(* PLC project LTAB4, Bombardier Transportation 1131-TOOL 3.1.0.1 *)
(* stored: companyURL www.kw-software.com, creationDateTime 2014-05-22T08:06:31, version 1400738791, modificationDateTime 2014-05-22T08:06:31 *)

FUNCTION_BLOCK DBC_PV_MtFanCtrl
  VAR_INPUT
    DBC_PV_X_ColStep : INT;
  END_VAR
  VAR_OUTPUT
    DBC_PV_C_Fan1Lo : BOOL;
    DBC_PV_C_Fan1Hi : BOOL;
    DBC_PV_C_Fan2Lo : BOOL;
    DBC_PV_C_Fan2Hi : BOOL;
    DBC_PV_C_Fan3Lo : BOOL;
    DBC_PV_C_Fan3Hi : BOOL;
  END_VAR
  VAR
    Enable : BOOL := TRUE;
    P_Fan1Lo_1 : INT := 3;
    P_Fan1Lo_2 : INT := 7;
    P_Fan1Hi : INT := 8;
    P_Fan2Lo_1 : INT := 4;
    P_Fan2Lo_2 : INT := 6;
    P_Fan2Hi_1 : INT := 7;
    P_Fan2Hi_2 : INT := 8;
    P_Fan3Lo : INT := 5;
    P_Fan3Hi_1 : INT := 6;
    P_Fan3Hi_2 : INT := 8;
  END_VAR

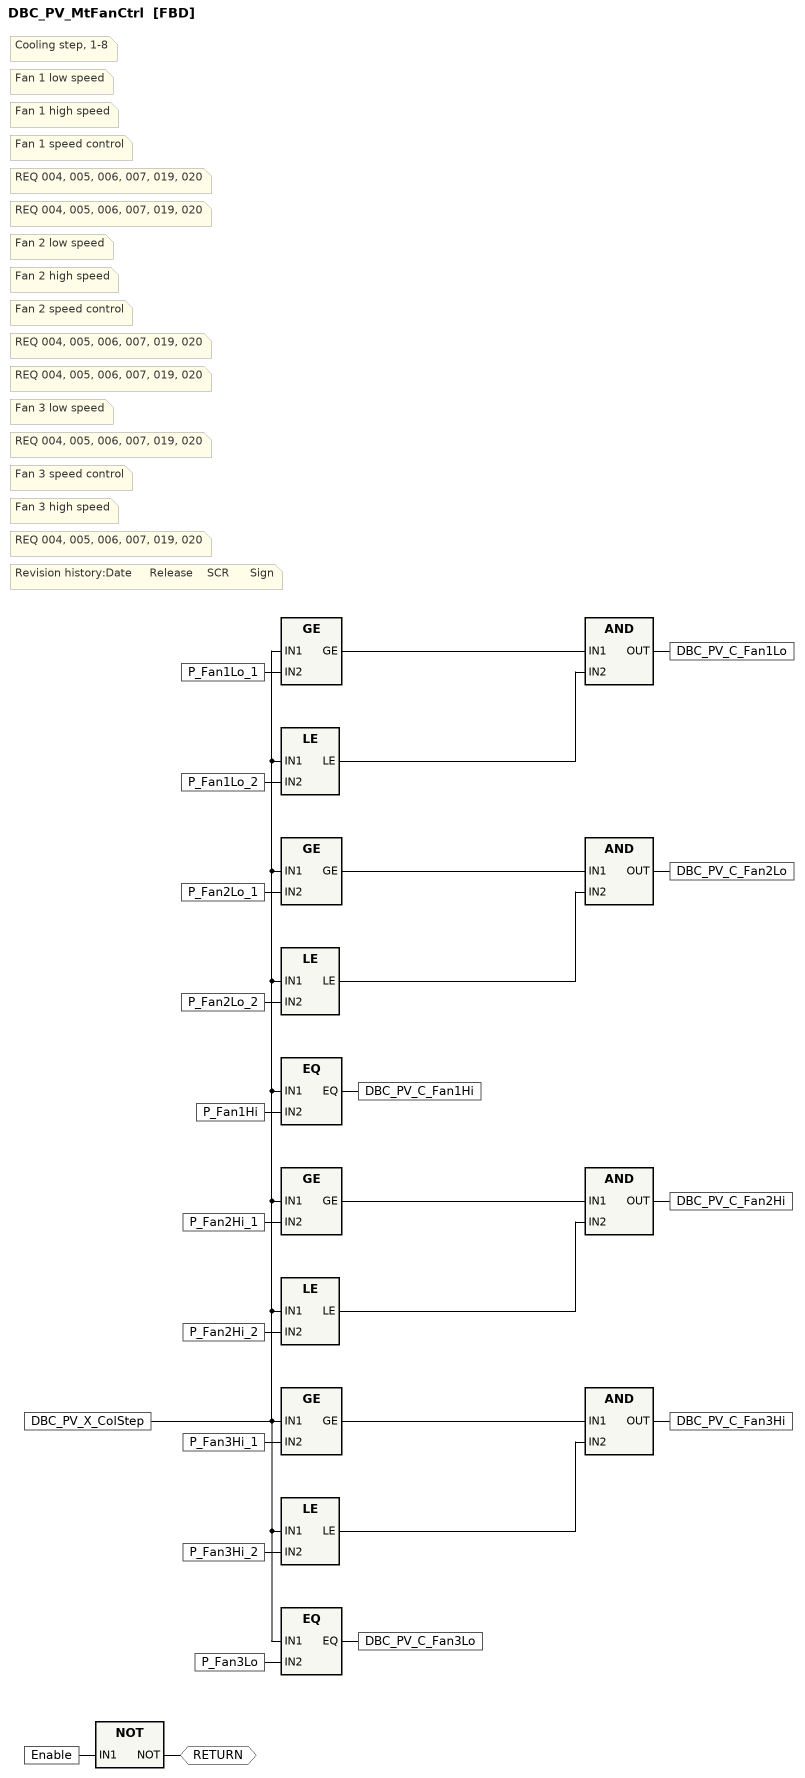
(* FBD diagram, written out as Structured Text *)
(* Fan 1 speed control *)
IF NOT Enable THEN RETURN; END_IF;
(* Cooling step, 1-8 *)
(* Fan 1 low speed *)
(* REQ 004, 005, 006, 007, 019, 020 *)
DBC_PV_C_Fan1Lo := DBC_PV_X_ColStep >= P_Fan1Lo_1 AND DBC_PV_X_ColStep <= P_Fan1Lo_2;
(* Fan 1 high speed *)
(* REQ 004, 005, 006, 007, 019, 020 *)
DBC_PV_C_Fan1Hi := DBC_PV_X_ColStep = P_Fan1Hi;
(* Fan 2 speed control *)
(* Fan 2 low speed *)
(* REQ 004, 005, 006, 007, 019, 020 *)
DBC_PV_C_Fan2Lo := DBC_PV_X_ColStep >= P_Fan2Lo_1 AND DBC_PV_X_ColStep <= P_Fan2Lo_2;
(* Fan 2 high speed *)
(* REQ 004, 005, 006, 007, 019, 020 *)
DBC_PV_C_Fan2Hi := DBC_PV_X_ColStep >= P_Fan2Hi_1 AND DBC_PV_X_ColStep <= P_Fan2Hi_2;
(* Fan 3 speed control *)
(* Fan 3 low speed *)
(* REQ 004, 005, 006, 007, 019, 020 *)
DBC_PV_C_Fan3Lo := DBC_PV_X_ColStep = P_Fan3Lo;
(* Fan 3 high speed *)
(* REQ 004, 005, 006, 007, 019, 020 *)
DBC_PV_C_Fan3Hi := DBC_PV_X_ColStep >= P_Fan3Hi_1 AND DBC_PV_X_ColStep <= P_Fan3Hi_2;
(* Revision history:

Date     Release    SCR      Sign *)
END_FUNCTION_BLOCK
